// TIA Portal V18 export
// export: Created 2026-06-05T07:40:24.9541532Z, ExportSetting WithDefaults, DisplayName Totally Integrated Automation Portal, DisplayVersion V18, DisplayName TIA Portal Openness, DisplayVersion V18, DisplayName TIA Portal Version Control Interface, DisplayVersion V18, DisplayName STEP 7 Professional, DisplayVersion V18, DisplayName STEP 7 Safety, DisplayVersion V18, DisplayName WinCC Professional, DisplayVersion V18
FUNCTION "FC_PLC1_Logic" : Void   // FC10, LAD
{ S7_Optimized_Access := 'TRUE' }
VERSION : 0.1
// stored: AutoNumber true, IsIECCheckEnabled false, SetENOAutomatically false, UDAEnableTagReadback false
BEGIN

REGION Network 1: Start Motor - Set bMotorRunning
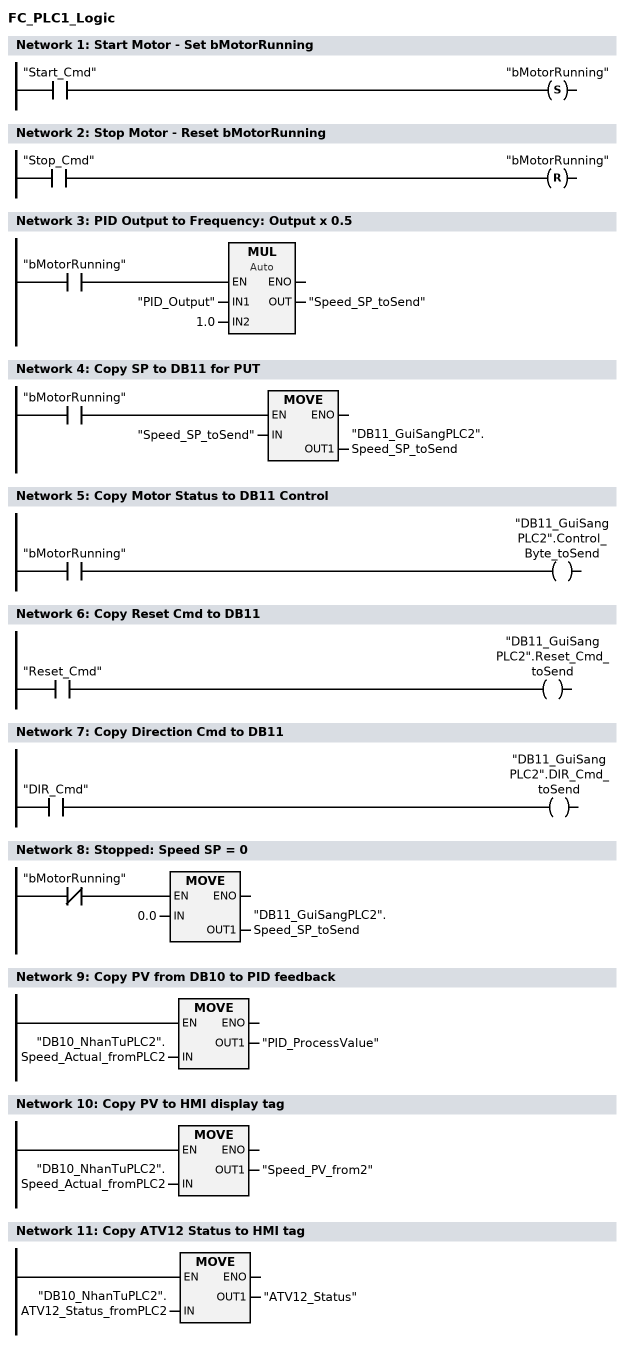
   RUNG wire#powerrail
      Contact( "Start_Cmd" )
      S_Coil( "bMotorRunning" )
   END_RUNG
   // the same network as SCL:
   IF "Start_Cmd" THEN "bMotorRunning" := TRUE; END_IF;
END_REGION

REGION Network 2: Stop Motor - Reset bMotorRunning
   RUNG wire#powerrail
      Contact( "Stop_Cmd" )
      R_Coil( "bMotorRunning" )
   END_RUNG
   // the same network as SCL:
   IF "Stop_Cmd" THEN "bMotorRunning" := FALSE; END_IF;
END_REGION

REGION Network 3: PID Output to Frequency: Output x 0.5
   RUNG wire#powerrail
      Contact( "bMotorRunning" )
      { S7_GenerateENO := "TRUE" } Mul(in1 := "PID_Output", in2 := 1.0, out => "Speed_SP_toSend")
   END_RUNG
   // the same network as SCL:
   IF "bMotorRunning" THEN "Speed_SP_toSend" := "PID_Output" * 1.0; END_IF;
END_REGION

REGION Network 4: Copy SP to DB11 for PUT
   RUNG wire#powerrail
      Contact( "bMotorRunning" )
      { S7_GenerateENO := "TRUE" } Move(in := "Speed_SP_toSend", out1 => "DB11_GuiSangPLC2".Speed_SP_toSend)
   END_RUNG
   // the same network as SCL:
   IF "bMotorRunning" THEN "DB11_GuiSangPLC2".Speed_SP_toSend := "Speed_SP_toSend"; END_IF;
END_REGION

REGION Network 5: Copy Motor Status to DB11 Control
   RUNG wire#powerrail
      Contact( "bMotorRunning" )
      Coil( "DB11_GuiSangPLC2".Control_Byte_toSend )
   END_RUNG
   // the same network as SCL:
   "DB11_GuiSangPLC2".Control_Byte_toSend := "bMotorRunning";
END_REGION

REGION Network 6: Copy Reset Cmd to DB11
   RUNG wire#powerrail
      Contact( "Reset_Cmd" )
      Coil( "DB11_GuiSangPLC2".Reset_Cmd_toSend )
   END_RUNG
   // the same network as SCL:
   "DB11_GuiSangPLC2".Reset_Cmd_toSend := "Reset_Cmd";
END_REGION

REGION Network 7: Copy Direction Cmd to DB11
   RUNG wire#powerrail
      Contact( "DIR_Cmd" )
      Coil( "DB11_GuiSangPLC2".DIR_Cmd_toSend )
   END_RUNG
   // the same network as SCL:
   "DB11_GuiSangPLC2".DIR_Cmd_toSend := "DIR_Cmd";
END_REGION

REGION Network 8: Stopped: Speed SP = 0
   RUNG wire#powerrail
      I_Contact( "bMotorRunning" )
      { S7_GenerateENO := "TRUE" } Move(in := 0.0, out1 => "DB11_GuiSangPLC2".Speed_SP_toSend)
   END_RUNG
   // the same network as SCL:
   IF NOT "bMotorRunning" THEN "DB11_GuiSangPLC2".Speed_SP_toSend := 0.0; END_IF;
END_REGION

REGION Network 9: Copy PV from DB10 to PID feedback
   RUNG wire#powerrail
      { S7_GenerateENO := "TRUE" } Move(in := "DB10_NhanTuPLC2".Speed_Actual_fromPLC2, out1 => "PID_ProcessValue")
   END_RUNG
   // the same network as SCL:
   "PID_ProcessValue" := "DB10_NhanTuPLC2".Speed_Actual_fromPLC2;
END_REGION

REGION Network 10: Copy PV to HMI display tag
   RUNG wire#powerrail
      { S7_GenerateENO := "TRUE" } Move(in := "DB10_NhanTuPLC2".Speed_Actual_fromPLC2, out1 => "Speed_PV_from2")
   END_RUNG
   // the same network as SCL:
   "Speed_PV_from2" := "DB10_NhanTuPLC2".Speed_Actual_fromPLC2;
END_REGION

REGION Network 11: Copy ATV12 Status to HMI tag
   RUNG wire#powerrail
      { S7_GenerateENO := "TRUE" } Move(in := "DB10_NhanTuPLC2".ATV12_Status_fromPLC2, out1 => "ATV12_Status")
   END_RUNG
   // the same network as SCL:
   "ATV12_Status" := "DB10_NhanTuPLC2".ATV12_Status_fromPLC2;
END_REGION
END_FUNCTION
